{attribute 'GeneratedUsingTerminal: ER2038-0001-0017'}
{attribute addProperty BoxType "ER2038-0001-0017"}
{attribute addProperty Id "InputAT %I*BOOL1"}
{attribute addProperty CRC "2198356929"}
{attribute addProperty Size "1"}
TYPE Diag_Channel_830843C1 EXTENDS InputBase_8311D824 :
STRUCT
	{attribute addProperty Name "Input"}
	Input AT %I* : BOOL;
END_STRUCT
END_TYPE

(* stored: Version 1.2.0.0, ProductVersion 3.1.4024.9
   DUT Diag_Channel_830843C1: Id {b071c7b3-4f89-44ac-8926-3472f76d8c81} *)
